{attribute 'GeneratedUsingTerminal: EL3773-0000-0017'}
{attribute addProperty BoxType "EL3773-0000-0017"}
{attribute addProperty Id "Cycle_CountAT %I*UINT2"}
{attribute addProperty CRC "2980656546"}
{attribute addProperty Size "2"}
TYPE AI_Sample_Count_B1A935A2 :
STRUCT
	{attribute addProperty Name "Cycle_Count"}
	Cycle_Count AT %I* : UINT;
END_STRUCT
END_TYPE

(* stored: Version 1.2.0.0, ProductVersion 3.1.4024.9
   DUT AI_Sample_Count_B1A935A2: Id {c0777052-32f6-4eba-a72b-b3a9371a8afc} *)
